# EPICS substitutions: db/Beckhoff_9XXX/ecmcEL9512.substitutions
file "ecmcEcSlave.template"
{
  pattern {}
          {}
}

file "ecmcEL95XX-chX.template"
{
  pattern {}
          {}
}
